FUNCTION_BLOCK PressureSensorScalingHandler
VAR_INPUT
	reactorPressureSensor : INT;
END_VAR
VAR_OUTPUT
	PressureScaledValue : INT;
END_VAR
VAR
END_VAR


// Scale analog pressure
PressureScaledValue := F_AnalogScale(AnalogInputRawValue := reactorPressureSensor, MaxAnalogValue := 1000);

END_FUNCTION_BLOCK

(* stored: Version 1.1.0.1, ProductVersion 3.1.4024.9
   POU PressureSensorScalingHandler: Id {6fd29d96-6b31-457b-8b2a-d64db9a9e64b}, SpecialFunc None *)
